// Mitsubishi GX Works2 project: 2026_01_21_PASSIVITY_AUTO_v2   PLC: Q03UDV

PROGRAM MAIN
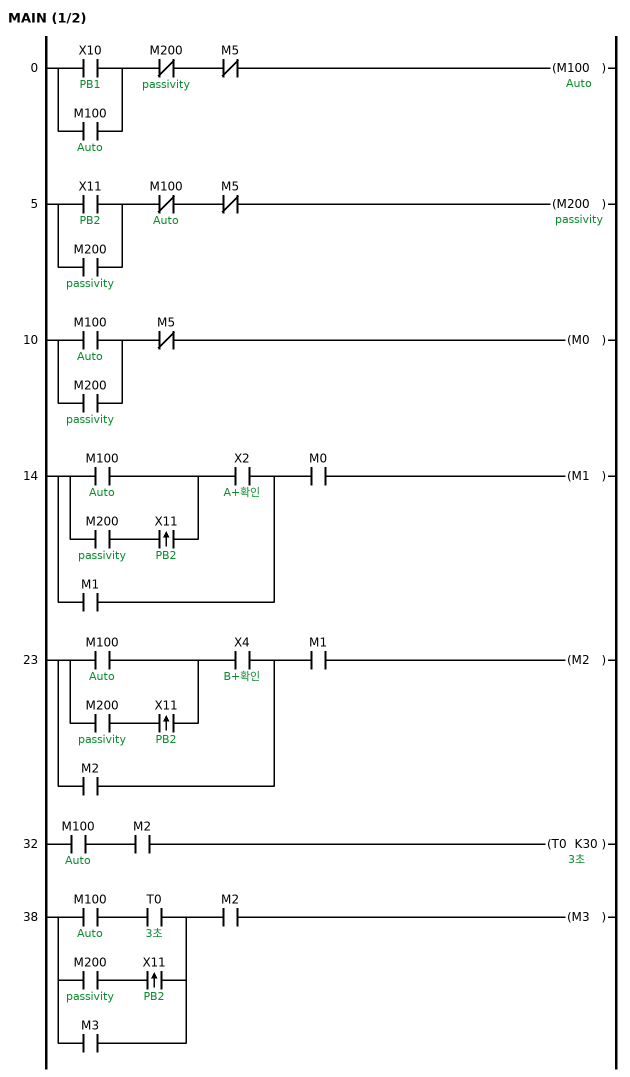
0     LD      X10  ; PB1
      OR      M100  ; Auto
      ANI     M200  ; passivity
      ANI     M5
      OUT     M100  ; Auto
5     LD      X11  ; PB2
      OR      M200  ; passivity
      ANI     M100  ; Auto
      ANI     M5
      OUT     M200  ; passivity
10    LD      M100  ; Auto
      OR      M200  ; passivity
      ANI     M5
      OUT     M0
14    LD      M100  ; Auto
      LD      M200  ; passivity
      ANDP    X11  ; PB2
      ORB
      AND     X2  ; A+확인
      OR      M1
      AND     M0
      OUT     M1
23    LD      M100  ; Auto
      LD      M200  ; passivity
      ANDP    X11  ; PB2
      ORB
      AND     X4  ; B+확인
      OR      M2
      AND     M1
      OUT     M2
32    LD      M100  ; Auto
      AND     M2
      OUT     T0 K30  ; 3초
38    LD      M100  ; Auto
      AND     T0  ; 3초
      LD      M200  ; passivity
      ANDP    X11  ; PB2
      ORB
      OR      M3
      AND     M2
      OUT     M3
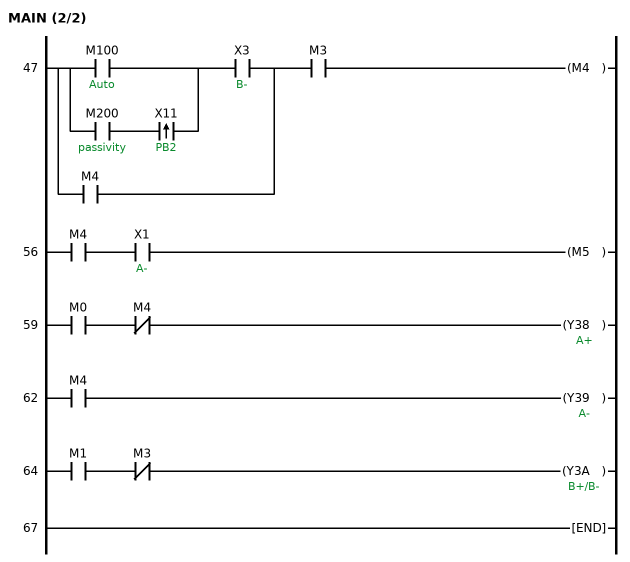
47    LD      M100  ; Auto
      LD      M200  ; passivity
      ANDP    X11  ; PB2
      ORB
      AND     X3  ; B-
      OR      M4
      AND     M3
      OUT     M4
56    LD      M4
      AND     X1  ; A-
      OUT     M5
59    LD      M0
      ANI     M4
      OUT     Y38  ; A+
62    LD      M4
      OUT     Y39  ; A-
64    LD      M1
      ANI     M3
      OUT     Y3A  ; B+/B-
67    END
END_PROGRAM
